PROGRAM ControlFBD
VAR
	qxLampStarted	AT %Q* : BOOL;
	qxSliderAout 	AT %Q* : BOOL; 
	qxSliderAin 	AT %Q* : BOOL; 
	qxSliderBout 	AT %Q* : BOOL; 
	qxSliderBin 	AT %Q* : BOOL; 
	qxDrillDown 	AT %Q* : BOOL;
	qxDrillUp		AT %Q* : BOOL;
	qxLampEmStopOk	AT %Q* : BOOL;
	qxLampSafetyOk  AT %Q* : BOOL;
	qxLampHomePos   AT %Q* : BOOL;
	
	
	ixButtonStart	AT %I* : BOOL;
	ixButtonStop	AT %I* : BOOL;
	ixSliderAout	AT %I* : BOOL;
	ixSliderAin		AT %I* : BOOL;
	ixSliderBout	AT %I* : BOOL;
	ixSliderBin		AT %I* : BOOL;
	ixDrillUp		AT %I* : BOOL;
	ixDrillDown		AT %I* : BOOL;

	ixAuto			AT %I* : BOOL;
	ixBtn1EmStopOk	AT %I* : BOOL;
	ixBtn2EmStopOk	AT %I* : BOOL;	
	ixSafety1StopOk	AT %I* : BOOL;
	ixSafety2StopOk	AT %I* : BOOL;	
	ixBtnReset		AT %I* : BOOL;
	ixBtnAout		AT %I* : BOOL;
	ixBtnAin		AT %I* : BOOL;
	ixBtnBout		AT %I* : BOOL;
	ixBtnBin		AT %I* : BOOL;
	ixBtnDrillOut	AT %I* : BOOL;
	ixBtnDrillIn	AT %I* : BOOL;
    
	mxEmStopReady: BOOL;
	mxEmStopOk: BOOL;
	fbBlink : BLINK;
    mxBlink : BOOL;
	mxSafetyReady: BOOL;
	mxSafetyStopOk: BOOL;
	mxManRunOk: BOOL;
	mxAutoModeReady: BOOL;
	mxCycleStopActivated: BOOL;
	mxAutoRunOk: BOOL;
	BLINK_0: BLINK;
	mxCycleStop: BOOL;
END_VAR
VAR_INPUT
	mxAutoAout: BOOL;
	mxAutoAin: BOOL;
	mxAutoDrillOut: BOOL;
	mxAutoDrillUp: BOOL;
	mxAutoBin: BOOL;
	mxAutoBout: BOOL;
	mxAutoDrillDown: BOOL;
END_VAR

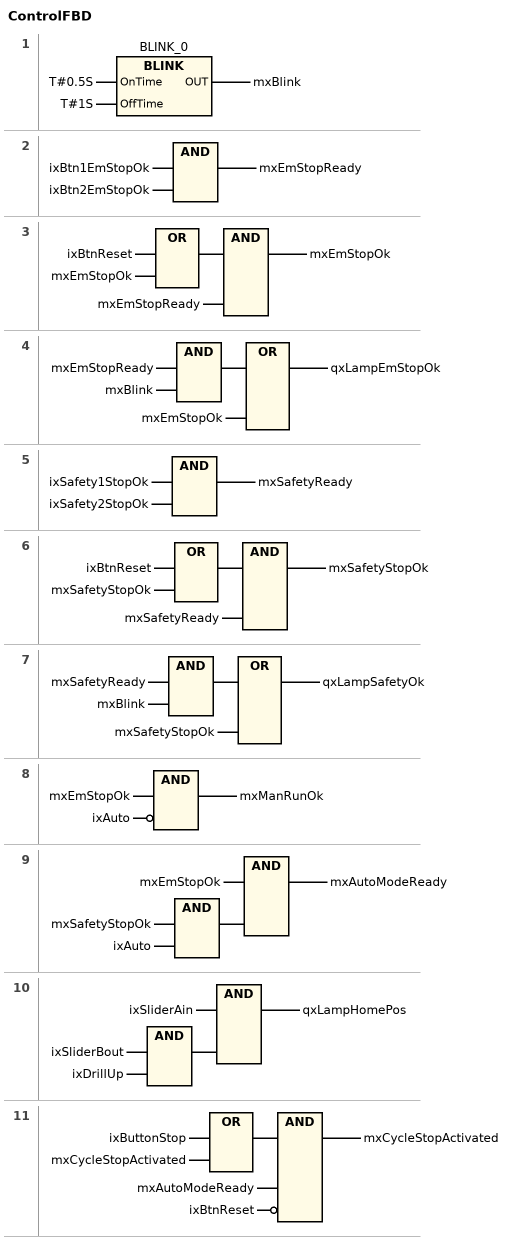
// NETWORK 1
BLINK_0(OnTime := T#0.5S, OffTime := T#1S); // BLINK
mxBlink := BLINK_0.OUT;

// NETWORK 2
mxEmStopReady := ixBtn1EmStopOk AND ixBtn2EmStopOk;

// NETWORK 3
mxEmStopOk := (ixBtnReset OR mxEmStopOk) AND mxEmStopReady;

// NETWORK 4
qxLampEmStopOk := mxEmStopReady AND mxBlink OR mxEmStopOk;

// NETWORK 5
mxSafetyReady := ixSafety1StopOk AND ixSafety2StopOk;

// NETWORK 6
mxSafetyStopOk := (ixBtnReset OR mxSafetyStopOk) AND mxSafetyReady;

// NETWORK 7
qxLampSafetyOk := mxSafetyReady AND mxBlink OR mxSafetyStopOk;

// NETWORK 8
mxManRunOk := mxEmStopOk AND NOT ixAuto;

// NETWORK 9
mxAutoModeReady := mxEmStopOk AND (mxSafetyStopOk AND ixAuto);

// NETWORK 10
qxLampHomePos := ixSliderAin AND (ixSliderBout AND ixDrillUp);

// NETWORK 11
mxCycleStopActivated := (ixButtonStop OR mxCycleStopActivated) AND mxAutoModeReady AND NOT ixBtnReset;

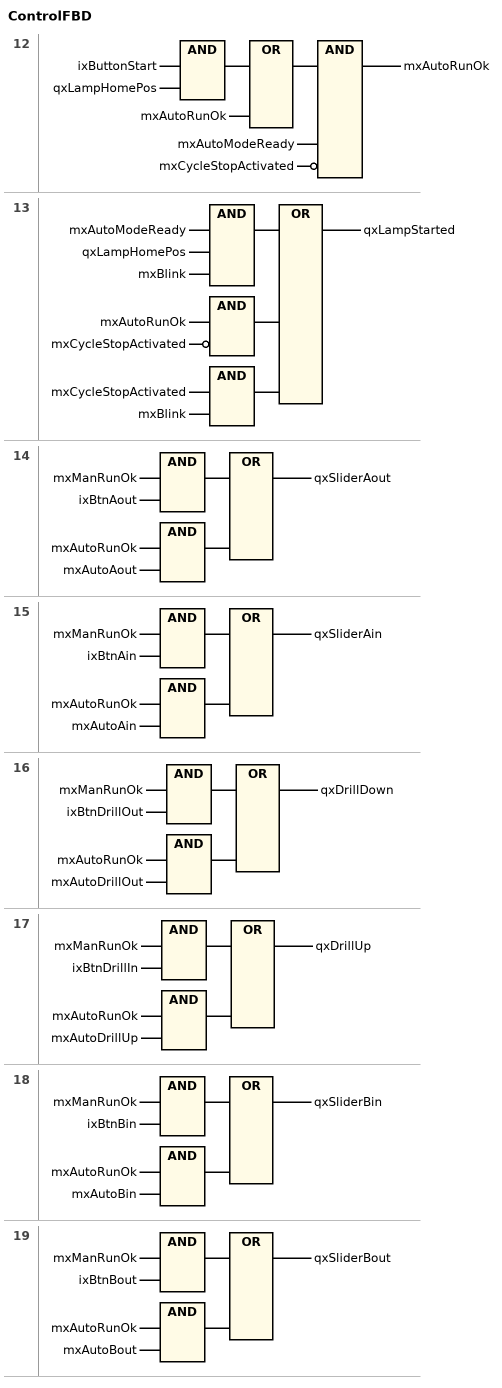
// NETWORK 12
mxAutoRunOk := (ixButtonStart AND qxLampHomePos OR mxAutoRunOk) AND mxAutoModeReady AND NOT mxCycleStopActivated;

// NETWORK 13
qxLampStarted := mxAutoModeReady AND qxLampHomePos AND mxBlink OR mxAutoRunOk AND NOT mxCycleStopActivated OR mxCycleStopActivated AND mxBlink;

// NETWORK 14
qxSliderAout := mxManRunOk AND ixBtnAout OR mxAutoRunOk AND mxAutoAout;

// NETWORK 15
qxSliderAin := mxManRunOk AND ixBtnAin OR mxAutoRunOk AND mxAutoAin;

// NETWORK 16
qxDrillDown := mxManRunOk AND ixBtnDrillOut OR mxAutoRunOk AND mxAutoDrillOut;

// NETWORK 17
qxDrillUp := mxManRunOk AND ixBtnDrillIn OR mxAutoRunOk AND mxAutoDrillUp;

// NETWORK 18
qxSliderBin := mxManRunOk AND ixBtnBin OR mxAutoRunOk AND mxAutoBin;

// NETWORK 19
qxSliderBout := mxManRunOk AND ixBtnBout OR mxAutoRunOk AND mxAutoBout;

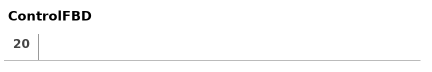
// NETWORK 20

END_PROGRAM

(* stored: Version 1.1.0.1
   POU ControlFBD: Id {441bf843-2f16-42db-a10b-d561aec11b1f}, SpecialFunc None *)
